FUNCTION_BLOCK StationSample EXTENDS Process
VAR_INPUT
	StateMachine : IPmlStateMachine;
END_VAR
VAR_OUTPUT
END_VAR
VAR
	_OperationTime : TIME := T#1S;
	Operation : ton;
	State: INT;
END_VAR

IF _isProcess THEN
	;
ELSE
	CASE State OF
		0:
			IF _HasMover THEN
				_Operating := TRUE;
				_Clear := FALSE;
				_Ready := FALSE;
				Operation.IN := TRUE;
				State := 1;
			END_IF
		1:
			IF Operation.Q THEN
				_Complete := TRUE;
				IF StationMovers = 0 THEN
					_HasMover := FALSE;
					Operation.IN := FALSE;
				END_IF
				State := 2;
			END_IF
		2:
			_Complete := FALSE;
			_Clear := TRUE;
			_Operating := FALSE;
			_Ready := TRUE;
			State := 0;
	END_CASE	
	Operation(PT := _OperationTime);
END_IF

IF StateMachine.GetCurrentState() = E_PMLState.ePMLState_Aborted THEN
	_Complete := FALSE;
	_Clear := TRUE;
	_Operating := FALSE;
	_Ready := TRUE;
	StationMovers := State := 0;
END_IF

SUPER^();
stInfo.StationProcessTime := _OperationTime;

PROPERTY TempPropTime : time
GET
TempPropTime := _OperationTime;
END_GET
SET
_OperationTime := TempPropTime;
END_SET
END_PROPERTY

END_FUNCTION_BLOCK

(* stored: Version 1.1.0.1, ProductVersion 3.1.4024.11
   POU StationSample: Id {2455d108-358d-48f3-a683-d527519dc5b8}, SpecialFunc None
   Property TempPropTime: Id {e0ccb7b2-ab4d-4401-a6ea-ec63ab2ed8d6}
   Get Get: Id {d09bc174-9f05-4e5a-bc80-e72251b6839f}
   Set Set: Id {cefc9927-2f03-41f9-b855-e64e1bbf9aa6} *)
